# B&R Automation Studio project SDCAxis
Automation Studio 4.5.2.102; Default project; technology packages: Acp10Arnc0 1.0.0

## Configuration Real

CPU 4PP065.0571-P74, AutomationRuntime D4.52, Build 4.1.2, Vc V4.25.0, Safety 1.6

### Task classes (Cpu.sw)
```
Cyclic#1 (cycle 2000 us, tolerance 0 us):
  SDCAxisCtr <- SDCAxisCtrl_X.prg
DataObjects: Arnc0sys
NcDataObjects: AxisInit <- AxisInit.dob, gAxis03a <- gAxis03obj.gAxis03a.dob, AxisApt <- AxisApt.dob, gAxis03i <- gAxis03obj.gAxis03i.dob
Binaries: TCData, Acp10map1, acp10cfg, Acp10map, arconfig, User, Role, sysconf, iomap, asfw, ashwd, arnc0cfg, Arnc0map
Libraries: Acp10sdc, Library, Acp10man, Acp10_MC, sys_lib, brsystem, asstring, powerlnk, asieccon, AsMath, Arnc0man, DataObj, AsArLog, FileIO, AsArProf, AsMem, Runtime, astime, Acp10par, NcGlobal, asiotime
```

### Hardware
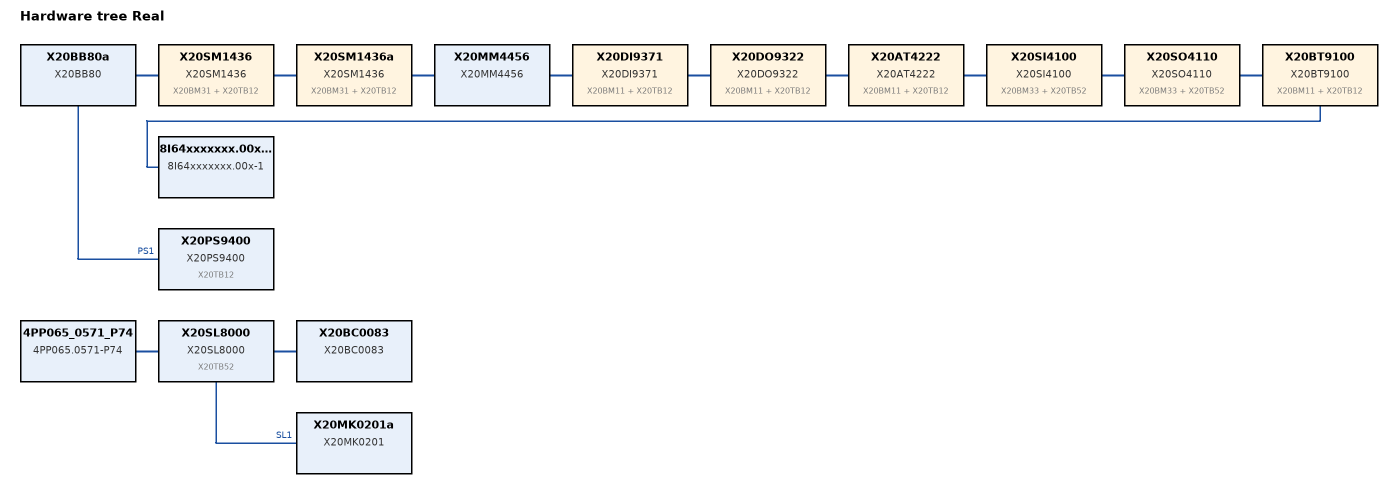
```
4PP065_0571_P74 : 4PP065.0571-P74 v1.1.2.0
  Connector IF4:
    EplInterfaceRedundant = 0
    EplEthInterfaceRedundant = 0
  Connector IF5:
    ActivateDevice = 1
    Mode = Manual
    InternetAddress = 10.0.1.14
    SubnetMask = 255.255.255.0
  ConfigurationID = labBR
  TimerDeviceType = EPLX2X
  TimerDevice = 4PP065_0571_P74.IF4
  TaskClassIdleTime = 2000
  Cyclic1Duration = 2000
  Cyclic1Tolerance = 0
  Cyclic1Output = 1
  Cyclic3Tolerance = 0
  VcObjectName = Visu
8I64xxxxxxx.00x-1 : 8I64xxxxxxx.00x-1 v1.3.9.1  [X2X1 -> X20BT9100.X2X1 [Cable Type=X2XCable, Length=10, Version=1.0.0.2]]
  BothEndSwitchesAreNormallyOpen_r1 = on
  QuickStopIsNormallyOpen_r1 = on
X20AT4222 : X20AT4222 v1.2.3.0  [SS1 -> X20TB12f.SS; SL -> X20BM11c.SL1]
X20BB80a : X20BB80 v1.0.2.0
X20BC0083 : X20BC0083 v2.7.0.0  [PLK1 -> X20SL8000.PLK2 (NodeNumber=2) [Cable Type=PowerlinkCable, Length=10, Version=1.0.0.2]; SL -> X20BB80a.SL1]
X20BM11a : X20BM11 v1.0.0.1  [X2X1 -> X20MM4456.X2X2]
X20BM11b : X20BM11 v1.0.0.1  [X2X1 -> X20BM11a.X2X2]
X20BM11c : X20BM11 v1.0.0.1  [X2X1 -> X20BM11b.X2X2]
X20BM11d : X20BM11 v1.0.0.1  [X2X1 -> X20BM33b.X2X2]
X20BM31a : X20BM31 v1.0.0.1  [X2X1 -> X20BB80a.IF1]
X20BM31b : X20BM31 v1.0.0.1  [X2X1 -> X20BM31a.X2X2]
X20BM33a : X20BM33 v1.0.0.4  [X2X1 -> X20BM11c.X2X2]
X20BM33b : X20BM33 v1.0.0.4  [X2X1 -> X20BM33a.X2X2]
X20BT9100 : X20BT9100 v1.0.3.0  [SS1 -> X20TB12g.SS; SL -> X20BM11d.SL1]
X20DI9371 : X20DI9371 v1.0.2.0  [SS1 -> X20TB12d.SS; SL -> X20BM11a.SL1]
X20DO9322 : X20DO9322 v1.0.3.0  [SS1 -> X20TB12e.SS; SL -> X20BM11b.SL1]
X20MK0201a : X20MK0201 v1.0.0.0  [SL -> X20SL8000.SL1]
X20MM4456 : X20MM4456 v1.1.5.0  [X2X1 -> X20BM31b.X2X2]
X20PS9400 : X20PS9400 v1.0.2.4  [SS1 -> X20TB12b.SS; PS -> X20BB80a.PS1]
X20SI4100 : X20SI4100 v1.10.1.1  [SS1 -> X20TB52b.SS; SL -> X20BM33a.SL1]
X20SL8000 : X20SL8000 v1.6.5.1  [PLK1 -> 4PP065_0571_P74.IF4 (NodeNumber=1) [Cable Type=PowerlinkCable, Length=10, Version=1.0.0.2]; PLK2 -> X20BC0083.PLK1 (NodeNumber=1) [Cable Type=PowerlinkCable, Length=10, Version=1.0.0.2]; SS1 -> X20TB52a.SS]
  SafeProject = SafeLOGIC-1
X20SM1436 : X20SM1436 v1.4.2.1  [SS1 -> X20TB12a.SS; SL -> X20BM31a.SL1]
X20SM1436a : X20SM1436 v1.4.2.1  [SS1 -> X20TB12c.SS; SL -> X20BM31b.SL1]
X20SO4110 : X20SO4110 v1.10.1.1  [SS1 -> X20TB52c.SS; SL -> X20BM33b.SL1]
  SafeLogicID = 2
  SafeModuleID = 3
X20TB12a : X20TB12 v1.0.0.0
X20TB12b : X20TB12 v1.0.0.0
X20TB12c : X20TB12 v1.0.0.0
X20TB12d : X20TB12 v1.0.0.0
X20TB12e : X20TB12 v1.0.0.0
X20TB12f : X20TB12 v1.0.0.0
X20TB12g : X20TB12 v1.0.0.0
X20TB52a : X20TB52 v1.0.0.1
X20TB52b : X20TB52 v1.0.0.1
X20TB52c : X20TB52 v1.0.0.1
```

### IoMap.iom - 4PP065_0571_P74/IoMap.iom
```iecst
VAR_CONFIG
	Cyclic#1.gAxis03_DrvIf.iLifeCnt AT %IB."8I64xxxxxxx.00x-1".SDC_LifeCnt;
	Cyclic#1.gAxis03_DrvIf.iDrvOK AT %IX."8I64xxxxxxx.00x-1".ETAD_Input_Bool_02;
	Cyclic#1.gAxis03_DrvIf.oSetTime AT %QW."8I64xxxxxxx.00x-1".SDC_SetTime;
	Cyclic#1.gAxis03_DrvIf.oSetPos AT %QW."8I64xxxxxxx.00x-1".LFRD_Output;
	Cyclic#1.gAxis03_DiDoIf.iLifeCntDriveReady AT %IB."8I64xxxxxxx.00x-1".SDC_LifeCnt;
	Cyclic#1.gAxis03_DiDoIf.iLifeCntDriveEnable AT %IB."8I64xxxxxxx.00x-1".SDC_LifeCnt;
	Cyclic#1.gAxis03_DiDoIf.oDriveEnable AT %QX."8I64xxxxxxx.00x-1".CMDD_Output_Bool_00;
	Cyclic#1.gAxis03_ModuleOk AT %QX."8I64xxxxxxx.00x-1".CMDD_Output_Bool_01;
	Cyclic#1.gAxis03_ModuleOk AT %QX."8I64xxxxxxx.00x-1".CMDD_Output_Bool_02;
	Cyclic#1.gAxis03_ModuleOk AT %IX."8I64xxxxxxx.00x-1".ModuleOk;
	Cyclic#1.gAxis03_DiDoIf.oDriveEnable AT %QX."8I64xxxxxxx.00x-1".CMDD_Output_Bool_03;
	Cyclic#1.gAxis03_DiDoIf.iDriveReady AT %IX."8I64xxxxxxx.00x-1".ETAD_Input_Bool_02;
	::SDCAxisCtr:pwm_period AT %QW."X20MM4456".PeriodDurationPWM;
	::SDCAxisCtr:coil_pwm_value AT %QW."X20MM4456".PulseWidthCurrentPWM04;
	::SDCAxisCtr:axis_X.pwm_value AT %QW."X20MM4456".PulseWidthCurrentPWM01;
	::SDCAxisCtr:axis_X.reset_error AT %QX."X20MM4456".ClearError01;
	::SDCAxisCtr:axis_X.reset_counter AT %QX."X20MM4456".ResetCounter01;
	::SDCAxisCtr:axis_X.counter AT %IW."X20MM4456".Counter01;
	::SDCAxisCtr:coil_powered AT %IX."X20DI9371".DigitalInput01;
	::SDCAxisCtr:axis_X.endswitch_a_reached AT %IX."X20MM4456".StatusInput03;
	::SDCAxisCtr:axis_X.endswitch_b_reached AT %IX."X20MM4456".StatusInput04;
END_VAR
```

### Acp10cfg.ncc - 4PP065_0571_P74/Motion/Acp10cfg.ncc
```
NcConfiguration (Version=3.13.1, NcSwId=Acp10)
  ACP10CF1_typ:
    cnt_nettrc_rec_drive = 1500
    bufsize_trace_upload = 1200
    tc_nc_man_task = Cyclic #1
    glob_pv_as_ncobject = Yes
    ncsys_dl_broadcast = Yes
    ncsys_dl_acp_reset = Yes
    safemc_log_err_to_ax = Yes
    network_init:
      ncsw_init_execute = Yes
      automatic_execute = No
      node_nr_warning = Yes
      net_err_before_ncact = Yes
    nettrc:
      enter_parsecrec = Yes
      enter_ncaction = Yes
      save_ring_startidx = Yes
    cam_prof_download:
      cam_dat_dl_parallel = No
      tc_cam_dl_parallel = Task class for NC Manager task
    sdc_if[0]:
      if_name = SDC_IF1
      mc_broadcast_size = 800
      mc_broadcast_extdat = No
```

### Acp10map.ncm - 4PP065_0571_P74/Motion/Acp10map.ncm
```
NcMapping (NcSwId=Acp10, DisabledNodesAreHidden=False)
  NcObject gAxis03 (ModuleId=8I64xxxxxxx.00x-1, ModuleAddress=SDC_IF1.ST1, Type=ncAXIS, Channel=1, AcoposSimulation=Off, InitParameter=gAxis03i, AcoposParameter=gAxis03a, AdditionalData=CNC_Enabled="1" , Disabled=FALSE, ModuleDisabled=FALSE)
```

### Acp10map1.ncm - 4PP065_0571_P74/Motion/Acp10map1.ncm
```
NcMapping (NcSwId=ACP10, DisabledNodesAreHidden=False)
  NcObject AxisX (ModuleAddress=SDC_IF1.ST2, InterfaceType=SDC, Type=ncAXIS, Channel=1, AcoposSimulation=Off, InitParameter=gAxis03i, AcoposParameter=gAxis03a, AdditionalData=CNC_Enabled="1" , Disabled=FALSE, ModuleDisabled=FALSE)
  NcObject AxisY (ModuleAddress=SDC_IF1.ST3, InterfaceType=SDC, Type=ncAXIS, Channel=1, AcoposSimulation=Off, InitParameter=AxisInit, AcoposParameter=AxisApt, AdditionalData=CNC_Enabled="1" , Disabled=FALSE)
  NcObject AxisZ (ModuleAddress=SDC_IF1.ST4, InterfaceType=SDC, Type=ncAXIS, Channel=1, AcoposSimulation=Off, InitParameter=AxisInit, AcoposParameter=AxisApt, AdditionalData=CNC_Enabled="1" , Disabled=FALSE)
```

### Arnc0cfg.ncc - 4PP065_0571_P74/Motion/Arnc0cfg.ncc
```
NcConfiguration (Version=3.13.1, NcSwId=Arnc0)
  ARNC0CFG_typ:
    sampling_rate = 4000
    cnt_nettrc_rec_drive = 150
    bufsize_sys_trace = 16#00005000
    enable_mp_log = Yes
    tc_nc_man_task = Cyclic #1
    bg_load = 1
    glob_pv_as_ncobject = Yes
```

### Arnc0map.ncm - 4PP065_0571_P74/Motion/Arnc0map.ncm
```
NcMapping (NcSwId=Arnc0, DisabledNodesAreHidden=False)
  NcObject CNCsys (Type=ncCNCSYS, Channel=1, AcoposSimulation=Off, InitParameter=CncInit, Disabled=FALSE, ModuleDisabled=FALSE)
  NcObject CNC2 (Type=ncCNCSYS, Channel=2, AcoposSimulation=Off, Disabled=TRUE, ModuleDisabled=FALSE)
  NcObject CNC3 (Type=ncCNCSYS, Channel=3, AcoposSimulation=Off, Disabled=TRUE, ModuleDisabled=FALSE)
  NcObject CNC4 (Type=ncCNCSYS, Channel=4, AcoposSimulation=Off, Disabled=TRUE, ModuleDisabled=FALSE)
  NcObject CNC5 (Type=ncCNCSYS, Channel=5, AcoposSimulation=Off, Disabled=TRUE, ModuleDisabled=FALSE)
  NcObject CNC6 (Type=ncCNCSYS, Channel=6, AcoposSimulation=Off, Disabled=TRUE, ModuleDisabled=FALSE)
  NcObject CNC7 (Type=ncCNCSYS, Channel=7, AcoposSimulation=Off, Disabled=TRUE, ModuleDisabled=FALSE)
  NcObject CNC8 (Type=ncCNCSYS, Channel=8, AcoposSimulation=Off, Disabled=TRUE, ModuleDisabled=FALSE)
  NcObject CNC9 (Type=ncCNCSYS, Channel=9, AcoposSimulation=Off, Disabled=TRUE, ModuleDisabled=FALSE)
  NcObject CNC10 (Type=ncCNCSYS, Channel=10, AcoposSimulation=Off, Disabled=TRUE, ModuleDisabled=FALSE)
  NcObject CNC11 (Type=ncCNCSYS, Channel=11, AcoposSimulation=Off, Disabled=TRUE, ModuleDisabled=FALSE)
  NcObject CNC12 (Type=ncCNCSYS, Channel=12, AcoposSimulation=Off, Disabled=TRUE, ModuleDisabled=FALSE)
  NcObject CNC13 (Type=ncCNCSYS, Channel=13, AcoposSimulation=Off, Disabled=TRUE, ModuleDisabled=FALSE)
  NcObject CNC14 (Type=ncCNCSYS, Channel=14, AcoposSimulation=Off, Disabled=TRUE, ModuleDisabled=FALSE)
  NcObject CNC15 (Type=ncCNCSYS, Channel=15, AcoposSimulation=Off, Disabled=TRUE, ModuleDisabled=FALSE)
  NcObject CNC16 (Type=ncCNCSYS, Channel=16, AcoposSimulation=Off, Disabled=TRUE, ModuleDisabled=FALSE)
  NcObject CNC17 (Type=ncCNCSYS, Channel=17, AcoposSimulation=Off, Disabled=TRUE, ModuleDisabled=FALSE)
  NcObject CNC18 (Type=ncCNCSYS, Channel=18, AcoposSimulation=Off, Disabled=TRUE, ModuleDisabled=FALSE)
  NcObject CNC19 (Type=ncCNCSYS, Channel=19, AcoposSimulation=Off, Disabled=TRUE, ModuleDisabled=FALSE)
  NcObject CNC20 (Type=ncCNCSYS, Channel=20, AcoposSimulation=Off, Disabled=TRUE, ModuleDisabled=FALSE)
  NcObject CNC21 (Type=ncCNCSYS, Channel=21, AcoposSimulation=Off, Disabled=TRUE, ModuleDisabled=FALSE)
  NcObject CNC22 (Type=ncCNCSYS, Channel=22, AcoposSimulation=Off, Disabled=TRUE, ModuleDisabled=FALSE)
  NcObject CNC23 (Type=ncCNCSYS, Channel=23, AcoposSimulation=Off, Disabled=TRUE, ModuleDisabled=FALSE)
  NcObject CNC24 (Type=ncCNCSYS, Channel=24, AcoposSimulation=Off, Disabled=TRUE, ModuleDisabled=FALSE)
```

## Configuration Simulation

CPU , AutomationRuntime J4.25, Safety 1.10

### Task classes (Cpu.sw)
```
Cyclic#1 (cycle 2000 us, tolerance 0 us):
  SDCAxisCtr <- SDCAxisCtrl_X.prg
  ncsdcctrl <- ncsdcctrl.prg
DataObjects: Acp10sys
NcDataObjects: AxisApt <- AxisApt.dob, AxisInit <- AxisInit.dob, acp10etxen <- acp10etxen.dob, gAxis05a <- gAxis05obj.gAxis05a.dob, gAxis05i <- gAxis05obj.gAxis05i.dob
Binaries: TCData, ashwd, sysconf, asfw, arconfig, iomap, Acp10map, Acp10map1, arnc0cfg, acp10cfg
Libraries: AsIecCon, astime, Acp10sdc, Acp10man, Acp10par, NcGlobal, asstring, AsIOTime, Acp10_MC, brsystem, sys_lib, Runtime, Acp10sim, fileio, powerlnk, Library, AsBrStr
```

### Hardware
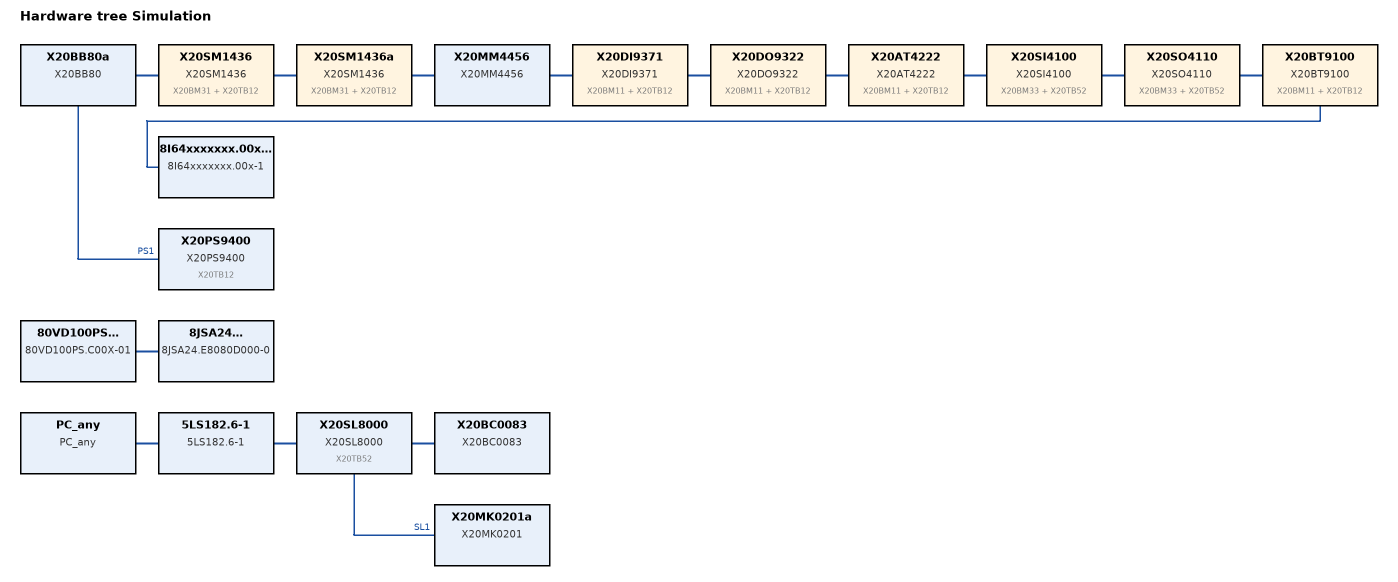
```
5LS182.6-1 : 5LS182.6-1 v1.3.0.0  [SL -> PC_any.SL1]
80VD100PS.C00X-01 : 80VD100PS.C00X-01 v2.3.0.1
8I64xxxxxxx.00x-1 : 8I64xxxxxxx.00x-1 v1.3.9.1  [X2X1 -> X20BT9100.X2X1 [Cable Type=X2XCable, Length=10, Version=1.0.0.2]]
  BothEndSwitchesAreNormallyOpen_r1 = on
  QuickStopIsNormallyOpen_r1 = on
8JSA24.E8080D000-0 : 8JSA24.E8080D000-0 v1.0.6.30  [MT -> 80VD100PS.C00X-01.MT1]
PC_any : PC_any v1.1.0.0 (OrderNumber=PC)
  ConfigurationID = SDCAxis_Simulation
  SystemTick = 2000
  Cyclic1Duration = 2000
  Cyclic1Tolerance = 0
  Cyclic1Output = 1
X20AT4222 : X20AT4222 v1.2.3.0  [SS1 -> X20TB12f.SS; SL -> X20BM11c.SL1]
X20BB80a : X20BB80 v1.0.2.0
X20BC0083 : X20BC0083 v2.7.0.0  [PLK2 -> X20SL8000.PLK2 (NodeNumber=2) [Cable Type=PowerlinkCable, Length=10, Version=1.0.0.2]; SL -> X20BB80a.SL1]
X20BM11a : X20BM11 v1.0.0.1  [X2X1 -> X20MM4456.X2X2]
X20BM11b : X20BM11 v1.0.0.1  [X2X1 -> X20BM11a.X2X2]
X20BM11c : X20BM11 v1.0.0.1  [X2X1 -> X20BM11b.X2X2]
X20BM11d : X20BM11 v1.0.0.1  [X2X1 -> X20BM33b.X2X2]
X20BM31a : X20BM31 v1.0.0.1  [X2X1 -> X20BB80a.IF1]
X20BM31b : X20BM31 v1.0.0.1  [X2X1 -> X20BM31a.X2X2]
X20BM33a : X20BM33 v1.0.0.4  [X2X1 -> X20BM11c.X2X2]
X20BM33b : X20BM33 v1.0.0.4  [X2X1 -> X20BM33a.X2X2]
X20BT9100 : X20BT9100 v1.0.3.0  [SS1 -> X20TB12g.SS; SL -> X20BM11d.SL1]
X20DI9371 : X20DI9371 v1.0.2.0  [SS1 -> X20TB12d.SS; SL -> X20BM11a.SL1]
X20DO9322 : X20DO9322 v1.0.3.0  [SS1 -> X20TB12e.SS; SL -> X20BM11b.SL1]
X20MK0201a : X20MK0201 v1.0.0.0  [SL -> X20SL8000.SL1]
X20MM4456 : X20MM4456 v1.1.5.0  [X2X1 -> X20BM31b.X2X2]
X20PS9400 : X20PS9400 v1.0.2.4  [SS1 -> X20TB12b.SS; PS -> X20BB80a.PS1]
X20SI4100 : X20SI4100 v1.10.1.1  [SS1 -> X20TB52b.SS; SL -> X20BM33a.SL1]
X20SL8000 : X20SL8000 v1.6.5.1  [PLK1 -> 5LS182.6-1.IF1 (NodeNumber=1) [Cable Type=PowerlinkCable, Length=10, Version=1.0.0.2]; PLK2 -> X20BC0083.PLK2 (NodeNumber=1) [Cable Type=PowerlinkCable, Length=10, Version=1.0.0.2]; SS1 -> X20TB52a.SS]
  SafeProject = SafeLOGIC-1
X20SM1436 : X20SM1436 v1.4.2.1  [SS1 -> X20TB12a.SS; SL -> X20BM31a.SL1]
X20SM1436a : X20SM1436 v1.4.2.1  [SS1 -> X20TB12c.SS; SL -> X20BM31b.SL1]
X20SO4110 : X20SO4110 v1.10.1.1  [SS1 -> X20TB52c.SS; SL -> X20BM33b.SL1]
  SafeLogicID = 2
  SafeModuleID = 3
X20TB12a : X20TB12 v1.0.0.0
X20TB12b : X20TB12 v1.0.0.0
X20TB12c : X20TB12 v1.0.0.0
X20TB12d : X20TB12 v1.0.0.0
X20TB12e : X20TB12 v1.0.0.0
X20TB12f : X20TB12 v1.0.0.0
X20TB12g : X20TB12 v1.0.0.0
X20TB52a : X20TB52 v1.0.0.1
X20TB52b : X20TB52 v1.0.0.1
X20TB52c : X20TB52 v1.0.0.1
```

### IOMap.iom - PC_any/IOMap.iom
```iecst
VAR_CONFIG
	::SDCAxisCtr:pwm_period AT %QW."X20MM4456".PeriodDurationPWM;
	::SDCAxisCtr:coil_pwm_value AT %QW."X20MM4456".PulseWidthCurrentPWM04;
	::SDCAxisCtr:axis_X.pwm_value AT %QW."X20MM4456".PulseWidthCurrentPWM01;
	::SDCAxisCtr:axis_X.reset_error AT %QX."X20MM4456".ClearError01;
	::SDCAxisCtr:axis_X.reset_counter AT %QX."X20MM4456".ResetCounter01;
	::SDCAxisCtr:axis_X.counter AT %IW."X20MM4456".Counter01;
	::SDCAxisCtr:axis_X.endswitch_a_reached AT %IX."X20MM4456".StatusInput03; (*Logical condition input 01=Motor 01:A*)
	::SDCAxisCtr:axis_X.endswitch_b_reached AT %IX."X20MM4456".StatusInput04; (*Logical condition input 02=Motor 01:B*)
	::SDCAxisCtr:coil_powered AT %IX."X20DI9371".DigitalInput01;
	Cyclic#1.gAxis03_DrvIf.iLifeCnt AT %IB."8I64xxxxxxx.00x-1".SDC_LifeCnt;
	Cyclic#1.gAxis03_DrvIf.iDrvOK AT %IX."8I64xxxxxxx.00x-1".ETAD_Input_Bool_02;
	Cyclic#1.gAxis03_DrvIf.oSetTime AT %QW."8I64xxxxxxx.00x-1".SDC_SetTime;
	Cyclic#1.gAxis03_DrvIf.oSetPos AT %QW."8I64xxxxxxx.00x-1".LFRD_Output;
	Cyclic#1.gAxis03_DiDoIf.iLifeCntDriveReady AT %IB."8I64xxxxxxx.00x-1".SDC_LifeCnt;
	Cyclic#1.gAxis03_DiDoIf.iLifeCntDriveEnable AT %IB."8I64xxxxxxx.00x-1".SDC_LifeCnt;
	Cyclic#1.gAxis03_DiDoIf.oDriveEnable AT %QX."8I64xxxxxxx.00x-1".CMDD_Output_Bool_00;
	Cyclic#1.gAxis03_ModuleOk AT %QX."8I64xxxxxxx.00x-1".CMDD_Output_Bool_01;
	Cyclic#1.gAxis03_ModuleOk AT %QX."8I64xxxxxxx.00x-1".CMDD_Output_Bool_02;
	Cyclic#1.gAxis03_ModuleOk AT %IX."8I64xxxxxxx.00x-1".ModuleOk;
	Cyclic#1.gAxis03_DiDoIf.oDriveEnable AT %QX."8I64xxxxxxx.00x-1".CMDD_Output_Bool_03;
	Cyclic#1.gAxis03_DiDoIf.iDriveReady AT %IX."8I64xxxxxxx.00x-1".ETAD_Input_Bool_02;
	      Cyclic#1.gAxis05_DrvIf.iLifeCnt AT %IB."X20SM1436".LifeCnt;
	      Cyclic#1.gAxis05_DrvIf.iDrvOK AT %IX."X20SM1436".DrvOk01;
	      Cyclic#1.gAxis05_DrvIf.oBoostCurrent AT %QX."X20SM1436".BoostCurrent01;
	      Cyclic#1.gAxis05_DrvIf.oStandStillCurrent AT %QX."X20SM1436".StandstillCurrent01;
	      Cyclic#1.gAxis05_DrvIf.oSetTime AT %QW."X20SM1436".SetTime01;
	      Cyclic#1.gAxis05_MotorStep0 AT %QW."X20SM1436".Motor1Step0;
	      Cyclic#1.gAxis05_DiDoIf.iLifeCntDriveEnable AT %IB."X20SM1436".LifeCnt;
	      Cyclic#1.gAxis05_DiDoIf.iLifeCntDriveReady AT %IB."X20SM1436".LifeCnt;
	      Cyclic#1.gAxis05_DiDoIf.iDriveReady AT %IX."X20SM1436".DrvOk01;
	      Cyclic#1.gAxis05_DiDoIf.oDriveEnable AT %QX."X20SM1436".DriveEnable01;
	      Cyclic#1.gAxis05_EncIf1.iLifeCnt AT %IB."X20SM1436".LifeCnt;
	      Cyclic#1.gAxis05_EncIf1.iEncOK AT %IX."X20SM1436".EncOk01;
	      Cyclic#1.gAxis05_EncIf1.iActPos AT %IW."X20SM1436".ActPos01;
	      Cyclic#1.gAxis05_EncIf1.iRefPulsePos AT %IW."X20SM1436".RefPulsePos01;
	      Cyclic#1.gAxis05_EncIf1.iRefPulseCnt AT %IB."X20SM1436".RefPulseCnt01;
	      Cyclic#1.gAxis05_EncIf1.iActTime AT %IW."X20SM1436".ActTime01;
END_VAR
```

### Acp10cfg.ncc - PC_any/Motion/Acp10cfg.ncc
```
NcConfiguration (Version=3.13.1, NcSwId=Acp10)
  ACP10CF1_typ:
    cnt_nettrc_rec_drive = 150
    bufsize_trace_upload = 1200
    tc_nc_man_task = Cyclic #1
    glob_pv_as_ncobject = Yes
    ncsys_dl_broadcast = Yes
    ncsys_dl_acp_reset = Yes
    safemc_log_err_to_ax = Yes
    network_init:
      ncsw_init_execute = Yes
      automatic_execute = No
      node_nr_warning = Yes
      net_err_before_ncact = Yes
    nettrc:
      enter_parsecrec = Yes
      enter_ncaction = Yes
      save_ring_startidx = No
    cam_prof_download:
      cam_dat_dl_parallel = No
      tc_cam_dl_parallel = Task class for NC Manager task
    sdc_if[0]:
      if_name = SDC_IF1
      mc_broadcast_size = 800
      mc_broadcast_extdat = No
```

### Acp10map.ncm - PC_any/Motion/Acp10map.ncm
```
NcMapping (NcSwId=Acp10)
  NcObject gAxis04 (ModuleId=8I64xxxxxxx.00x-1, ModuleAddress=SDC_IF1.ST2, Type=ncAXIS, Channel=1, AcoposSimulation=Off, InitParameter=gAxis03i, AcoposParameter=gAxis03a, AdditionalData=CNC_Enabled="1" , Disabled=FALSE, ModuleDisabled=FALSE)
  NcObject gAxis05 (ModuleId=X20SM1436, ModuleAddress=SDC_IF1.ST3, Type=ncAXIS, Channel=1, AcoposSimulation=Off, InitParameter=gAxis05i, AcoposParameter=gAxis05a, Disabled=FALSE, ModuleDisabled=FALSE)
  NcObject X20SM1436a_ncAXIS1 (ModuleId=X20SM1436a, ModuleAddress=SDC_IF1.ST4, Type=ncAXIS, Channel=1, AcoposSimulation=Off, Disabled=TRUE, ModuleDisabled=FALSE)
```

### Acp10map1.ncm - PC_any/Motion/Acp10map1.ncm
```
NcMapping (NcSwId=ACP10, DisabledNodesAreHidden=False)
  NcObject MyLittleAxis (ModuleAddress=SDC_IF1.ST1, InterfaceType=SDC, Type=ncAXIS, Channel=1, AcoposSimulation=Off, InitParameter=MyLittleIn, AcoposParameter=MyLittleAp, Disabled=FALSE, ModuleDisabled=FALSE)
```

### Arnc0cfg.ncc - PC_any/Motion/Arnc0cfg.ncc
```
NcConfiguration (Version=1.45.0, NcSwId=ARNC0)
  ARNC0CFG_typ:
    sampling_rate = 4000
    cnt_nettrc_rec_drive = 150
    bufsize_sys_trace = 16#00005000
    enable_mp_log = Yes
    tc_nc_man_task = Cyclic #1
    bg_load = 1
    glob_pv_as_ncobject = Yes
```

## Logical view

Binary libraries used (declarations not repeated): Runtime, OPERATOR, AsIecCon, astime, Acp10sdc 3.13.1, Acp10man 3.13.1, Acp10par 3.13.1, NcGlobal 3.13.1, asstring, AsIOTime, Acp10_MC 3.13.1, brsystem, sys_lib, Acp10sim 3.13.1, AsMath, Arnc0man 3.13.0, DataObj, AsArLog, FileIO, AsArProf, AsMem, AsBrStr

### Global.var - Global variables
```iecst
VAR
	AxisX : ACP10AXIS_typ := (0);
	AxisX_EncIf : SdcEncIf16_typ := (0);
	AxisX_DrvIf : SdcDrvIf16_typ := (0);
	AxisX_DiDoIf : SdcDiDoIf_typ := (0);
	AxisX_HW : SdcHwCfg_typ := (0);
	gAxis01 : ACP10AXIS_typ := (0);
	gAxis02 : ACP10AXIS_typ := (0);
	gAxisTest : ACP10AXIS_typ := (0);
	gAxisTest_HW : SdcHwCfg_typ := (0);
	gAxisTest_DrvIf : SdcDrvIf16_typ := (0);
	gAxisTest_DiDoIf : SdcDiDoIf_typ := (0);
	gAxisTest_ModuleOk : BOOL := 0;
	gAxis03 : ACP10AXIS_typ := (0);
	gAxis03_HW : SdcHwCfg_typ := (0);
	gAxis03_DrvIf : SdcDrvIf16_typ := (0);
	gAxis03_DiDoIf : SdcDiDoIf_typ := (0);
	gAxis03_ModuleOk : BOOL := 0;
	CNCsys : ARNC0CNC_typ;
	gAxis04 : ACP10AXIS_typ := (0);
	gAxis05 : ACP10AXIS_typ := (0);
	gAxis05_HW : SdcHwCfg_typ := (0);
	gAxis05_DrvIf : SdcDrvIf16_typ := (0);
	gAxis05_EncIf1 : SdcEncIf16_typ := (0);
	gAxis05_DiDoIf : SdcDiDoIf_typ := (0);
	gAxis05_MotorStep0 : INT := 0;
	coil_powered : BOOL := FALSE;
	coil_pwm_value : INT := 0;
	fb_regulator : FB_Regulator;
	pwm_period : UINT := 0;
	axis_X : FB_Axis := (0);
	iPosHwEnd : BOOL := FALSE;
	iNegHwEnd : BOOL := FALSE;
	iActPos : USINT := 0;
	oSetPos : USINT := 0;
END_VAR
```

### Package Logical/Libraries - Global libraries

### Library Logical/Libraries/Library (ANSIC)

#### Library.fun
```iecst
FUNCTION_BLOCK FB_Motor (*TODO: Add your comment here*) (*$GROUP=User,$CAT=User,$GROUPICON=User.png,$CATICON=User.png*)
	VAR_INPUT
		in : REAL;
	END_VAR
	VAR_OUTPUT
		out_w : REAL;
		out_phi : REAL;
	END_VAR
	VAR
		k_e : REAL;
		T_m : REAL;
		dt : REAL;
		integrator : FB_Integrator;
		integrator_phi : FB_Integrator;
	END_VAR
END_FUNCTION_BLOCK

FUNCTION_BLOCK FB_Integrator (*TODO: Add your comment here*) (*$GROUP=User,$CAT=User,$GROUPICON=User.png,$CATICON=User.png*)
	VAR_INPUT
		in : REAL;
		dt : REAL;
	END_VAR
	VAR_OUTPUT
		out : REAL;
	END_VAR
	VAR
		state : REAL := 0.0;
	END_VAR
END_FUNCTION_BLOCK

FUNCTION_BLOCK FB_Controller (* *) (*$GROUP=User,$CAT=User,$GROUPICON=User.png,$CATICON=User.png*)
	VAR_INPUT
		in : REAL;
	END_VAR
	VAR_OUTPUT
		out : REAL;
	END_VAR
	VAR
		k_i : REAL;
		sum : REAL;
		k_p : REAL;
		dt : REAL;
		max_abs_value : REAL;
		integrator : FB_Integrator;
		last_sum : REAL;
	END_VAR
END_FUNCTION_BLOCK

FUNCTION_BLOCK FB_Endswitch (*TODO: Add your comment here*) (*$GROUP=User,$CAT=User,$GROUPICON=User.png,$CATICON=User.png*)
	VAR_INPUT
		in : REAL;
		neg_value : REAL;
		pos_value : REAL;
	END_VAR
	VAR_OUTPUT
		neg_reached : BOOL;
		pos_reached : BOOL;
	END_VAR
END_FUNCTION_BLOCK

FUNCTION_BLOCK FB_Axis (*TODO: Add your comment here*) (*$GROUP=User,$CAT=User,$GROUPICON=User.png,$CATICON=User.png*)
	VAR_INPUT
		u : REAL;
		reset_error : BOOL;
		endswitch_a_reached : BOOL;
		endswitch_b_reached : BOOL;
		pwm_percentage : SINT;
	END_VAR
	VAR_OUTPUT
		reset_counter : BOOL;
		pwm_value : INT;
	END_VAR
	VAR_OUTPUT RETAIN
		counter : INT;
	END_VAR
	VAR_OUTPUT
		speed : REAL;
	END_VAR
	VAR
		i : INT;
		last_counter : INT;
		dir : BOOL;
		spid : REAL;
		k : INT;
	END_VAR
END_FUNCTION_BLOCK

{REDUND_ERROR} FUNCTION_BLOCK FB_Regulator (*TODO: Add your comment here*) (*$GROUP=User,$CAT=User,$GROUPICON=User.png,$CATICON=User.png*)
	VAR_INPUT
		e : REAL;
	END_VAR
	VAR_OUTPUT
		u : REAL;
	END_VAR
	VAR
		k_p : REAL;
		k_i : REAL;
		integrator : FB_Integrator;
		iyOld : REAL;
		max_abc_value : REAL := 24;
		dt : REAL;
		x : REAL;
	END_VAR
END_FUNCTION_BLOCK
```

#### FB_Motor.c
```c
#include <bur/plctypes.h>
#ifdef __cplusplus
	extern "C"
	{
#endif
	#include "Library.h"
#ifdef __cplusplus
	};
#endif
/* TODO: Add your comment here */
void FB_Motor(struct FB_Motor* inst)
{/*
	inst->integrator.in = (inst->u/inst->ke - inst->w) * (inst->dt/inst->Tm);
	FB_Integrator(&inst->integrator);
	inst->w = inst->integrator.out;
	inst->integrator.in = inst->w * inst->dt;
	FB_Integrator(&inst->integrator);
	inst->phi = inst->integrator.out;*/
}
```

#### FB_Controller.c
```c
#include <bur/plctypes.h>
#ifdef __cplusplus
	extern "C"
	{
#endif
	#include "Library.h"
#ifdef __cplusplus
	};
#endif

void FB_Controller(struct FB_Controller* inst)
{

}
```

#### FB_Integrator.c
```c
#include <bur/plctypes.h>
#ifdef __cplusplus
	extern "C"
	{
#endif
	#include "Library.h"
#ifdef __cplusplus
	};
#endif
/* TODO: Add your comment here */
void FB_Integrator(struct FB_Integrator* inst)
{
	inst->out = inst->dt * inst->in + inst->state;
	inst->state = inst->out;
}
```

#### FB_Endswitch.c
```c
#include <bur/plctypes.h>
#ifdef __cplusplus
	extern "C"
	{
#endif
	#include "Library.h"
#ifdef __cplusplus
	};
#endif
/* TODO: Add your comment here */
void FB_Endswitch(struct FB_Endswitch* inst)
{

}
```

#### FB_Axis.c
```c
#include <bur/plctypes.h>
#ifdef __cplusplus
	extern "C"
	{
#endif
	#include "Library.h"
#ifdef __cplusplus
	};
#endif
/* TODO: Add your comment here */
void FB_Axis(struct FB_Axis* inst)
{
	if (inst->endswitch_a_reached == 1 )
	{
		inst->dir = 1;
	}
	if (inst->endswitch_b_reached == 1 )
	{
		inst->dir = 0;
	}

	if(inst->dir == 1)
	{
		//inst->reset_counter = 0;
		inst->u = -inst->u;
		inst->pwm_value = (inst->u/24.0) * 32767;
	}
	if(inst->dir == 0)
	{
		//inst->reset_counter = 0;
		inst->pwm_value = (inst->u/24.0) * 32767;
	}
	if (inst->i == 1000)
	{
		inst->speed = (inst->counter - inst->last_counter)/2;
		inst->last_counter = inst->counter;
		inst->i = 0;
	}
	inst->spid = inst->speed;
	inst->i++;
}
```

#### FB_Regulator.c
```c
#include <bur/plctypes.h>
#ifdef __cplusplus
	extern "C"
	{
#endif
	#include "Library.h"
#ifdef __cplusplus
	};
#endif
/* TODO: Add your comment here */
void FB_Regulator(struct FB_Regulator* inst)
{
	float BON(float x)
		{
		if(x < 0)
		{
			if(x < -inst->max_abc_value)
				return -inst->max_abc_value;
			else
				return x;
		}
		else
		{
			if(x > inst->max_abc_value)
				return inst->max_abc_value;
			else
				return x;
		}

	}
	inst->integrator.in = inst->e * inst->k_i * inst->dt + inst->iyOld;
	FB_Integrator(&inst->integrator);
	inst->u = BON((BON(inst->e * inst->k_p) + inst->integrator.out));

	inst->iyOld = inst->u - (BON(inst->e * inst->k_p) + inst->integrator.out);
}
```

### Library Logical/Libraries/Library1 (ANSIC)

#### Library1.fun - Exported functions and function blocks
```iecst
{REDUND_ERROR} {REDUND_UNREPLICABLE} FUNCTION_BLOCK FB_Integrator (*TODO: Add your comment here*) (*$GROUP=User,$CAT=User,$GROUPICON=User.png,$CATICON=User.png*)
	VAR_INPUT
		in : {REDUND_UNREPLICABLE} REAL;
	END_VAR
	VAR_OUTPUT
		out : {REDUND_UNREPLICABLE} REAL;
	END_VAR
	VAR
		dt : {REDUND_UNREPLICABLE} REAL;
	END_VAR
END_FUNCTION_BLOCK

{REDUND_ERROR} {REDUND_UNREPLICABLE} FUNCTION_BLOCK FBMotor (*TODO: Add your comment here*) (*$GROUP=User,$CAT=User,$GROUPICON=User.png,$CATICON=User.png*)
	VAR_INPUT
		u : {REDUND_UNREPLICABLE} REAL;
	END_VAR
	VAR_OUTPUT
		w : {REDUND_UNREPLICABLE} REAL;
		phi : {REDUND_UNREPLICABLE} REAL;
	END_VAR
	VAR
		integrator : {REDUND_UNREPLICABLE} FB_Integrator;
		Tm : {REDUND_UNREPLICABLE} REAL;
		ke : {REDUND_UNREPLICABLE} REAL;
		dt : {REDUND_UNREPLICABLE} REAL;
	END_VAR
END_FUNCTION_BLOCK

{REDUND_ERROR} {REDUND_UNREPLICABLE} FUNCTION_BLOCK FB_Regulator (*TODO: Add your comment here*) (*$GROUP=User,$CAT=User,$GROUPICON=User.png,$CATICON=User.png*)
	VAR_INPUT
		e : {REDUND_UNREPLICABLE} REAL;
	END_VAR
	VAR_OUTPUT
		u : {REDUND_UNREPLICABLE} REAL;
	END_VAR
	VAR
		k_p : {REDUND_UNREPLICABLE} REAL;
		k_i : {REDUND_UNREPLICABLE} REAL;
		integrator : {REDUND_UNREPLICABLE} FB_Integrator;
		iyOld : {REDUND_UNREPLICABLE} REAL;
		max_abc_value : {REDUND_UNREPLICABLE} REAL;
		dt : {REDUND_UNREPLICABLE} REAL;
		x : {REDUND_UNREPLICABLE} REAL;
	END_VAR
END_FUNCTION_BLOCK
```

#### FB_Integrator.c
```c
#include <bur/plctypes.h>
#ifdef __cplusplus
	extern "C"
	{
#endif
	#include "Library1.h"
#ifdef __cplusplus
	};
#endif
/* TODO: Add your comment here */
void FB_Integrator(struct FB_Integrator* inst)
{
	inst->out = inst->in  + inst->out;

}
```

#### FBMotor.c
```c
#include <bur/plctypes.h>
#ifdef __cplusplus
	extern "C"
	{
#endif
	#include "Library1.h"
#ifdef __cplusplus
	};
#endif
/* TODO: Add your comment here */
void FBMotor(struct FBMotor* inst)
{
	inst->integrator.in = (inst->u/inst->ke - inst->w) * (inst->dt/inst->Tm);
	FB_Integrator(&inst->integrator);
	inst->w = inst->integrator.out;
	inst->integrator.in = inst->w * inst->dt;
	FB_Integrator(&inst->integrator);
	inst->phi = inst->integrator.out;
}
```

#### FB_Regulator.c
```c
#include <bur/plctypes.h>
#ifdef __cplusplus
	extern "C"
	{
#endif
	#include "Library1.h"
#ifdef __cplusplus
	};
#endif
/* TODO: Add your comment here */
void FB_Regulator(struct FB_Regulator* inst)
{
	float BON(float x)
	{
		if(x < 0)
		{
			if(x < -inst->max_abc_value)
				return -inst->max_abc_value;
			else
				return x;
		}
		else
		{
			if(x > inst->max_abc_value)
				return inst->max_abc_value;
			else
				return x;
		}

	}
	inst->integrator.in = inst->e * inst->k_i * inst->dt + inst->iyOld;
	FB_Integrator(&inst->integrator);
	inst->u = BON((BON(inst->e * inst->k_p) + inst->integrator.out));

	inst->iyOld = inst->u - (BON(inst->e * inst->k_p) + inst->integrator.out);
}
```

### Data object Logical/AxisApt (Apt)

#### AcpParTab.apt
```
AcoposParameterTable:
  Root Parameters:
    64201 = 4000 (Name=SERVO_V_MAX_OUTPUT, Unit=Units/s)  // Servo drive adjustment: Velocity at maximum output value
    109 = 24 (Name=SCALE_ENCOD_INCR)  // Encoder1: Encoder scaling: increments per encoder revolution
```

### Data object Logical/AxisInit (Ax)

#### AxInitAcp10.ax
```
InitParameter (Version=3.13.1, NcSwId=ACP10)
  ACP10AXIS_typ:
    dig_in:
      level:
        reference = ncACTIV_HI
        pos_hw_end = ncACTIV_HI
        neg_hw_end = ncACTIV_HI
        trigger1 = ncACTIV_HI
        trigger2 = ncACTIV_HI
    encoder_if:
      parameter:
        count_dir = ncSTANDARD
        scaling:
          load:
            units = 3000
            rev_motor = 1
    limit:
      parameter:
        v_pos = 7500.0
        v_neg = 7500.0
        a1_pos = 10000.0
        a2_pos = 10000.0
        a1_neg = 10000.0
        a2_neg = 10000.0
        t_jolt = 0.0
        t_in_pos = 0.0
        pos_sw_end = 8388607
        neg_sw_end = -8388608
        ds_warning = 500.0
        ds_stop = 50000.0
        a_stop = 1.0E+30
        dv_stop = 0.0
        dv_stop_mode = ncOFF
    controller:
      mode = ncPOSITION
      position:
        kv = 10.0
        tn = 0.0
        t_predict = 0.04
        t_total = 0.04
        p_max = 10000.0
        i_max = 0.0
      speed:
        kv = 2.0
        tn = 0.0
        t_filter = 0.0
        isq_filter1:
          type = ncOFF
          a0 = 0.0
          a1 = 0.0
          b0 = 0.0
          b1 = 0.0
          b2 = 0.0
          c0_par_id = 0
          c1_par_id = 0
        isq_filter2:
          type = ncOFF
          a0 = 0.0
          a1 = 0.0
          b0 = 0.0
          b1 = 0.0
          b2 = 0.0
          c0_par_id = 0
          c1_par_id = 0
        isq_filter3:
          type = ncOFF
          a0 = 0.0
          a1 = 0.0
          b0 = 0.0
          b1 = 0.0
          b2 = 0.0
          c0_par_id = 0
          c1_par_id = 0
      uf:
        type = ncLINEAR
        auto_config = ncMOTOR_PAR
        u0 = 0.0
        un = 0.0
        fn = 50.0
        k_f_slip = 0.0
      ff:
        torque_load = 0.0
        torque_pos = 0.0
        torque_neg = 0.0
        kv_torque = 0.0
        inertia = 0.0
        t_filter_a = 0.0
    move:
      stop:
        parameter[0]:
          decel_ramp = ncA_LIMIT
          controller = ncON
        parameter[1]:
          decel_ramp = ncA_LIMIT
          controller = ncON
        parameter[2]:
          decel_ramp = ncA_LIMIT
          controller = ncON
        parameter[3]:
          decel_ramp = ncA_LIMIT
          controller = ncON
        quickstop:
          decel_ramp = ncA_LIMIT
        drive_error:
          decel_ramp = ncA_LIMIT
      homing:
        parameter:
          s = 0
          v_switch = 6000.0
          v_trigger = 2000.0
          a = 10000.0
          mode = ncEND_SWITCH
          edge_sw = ncNEGATIVE
          start_dir = ncPOSITIVE
          trigg_dir = ncNEGATIVE
          ref_pulse = ncOFF
          fix_dir = ncOFF
          tr_s_block = 0.0
          torque_lim = 0.0
          ds_block = 0.0
          ds_stop = 0.0
      basis:
        parameter:
          v_pos = 4000.0
          v_neg = 4000.0
          a1_pos = 10000.0
          a2_pos = 10000.0
          a1_neg = 10000.0
          a2_neg = 10000.0
    message:
      text:
        parameter:
          format = ncBREAK
          columns = 80
          data_modul
```

### Data object Logical/acp10etxen (Ett)

- acp10etxen.ett (not shown)

### Package Logical/gAxis03obj - gAxis03obj

### Data object Logical/gAxis03obj/gAxis03a (Apt)

#### gAxis03a.apt
```
AcoposParameterTable:
  Root Parameters:
    230 = PCTRL_S_SET (Name=PCTRL_S_ACT_PARID)
    64201 = 546116.666666667 (Name=SERVO_V_MAX_OUTPUT)
```

### Data object Logical/gAxis03obj/gAxis03i (Ax)

#### gAxis03i.ax
```
InitParameter (Version=3.13.1, NcSwId=Acp10)
  ACP10AXIS_typ:
    dig_in:
      level:
        reference = ncACTIV_HI
        pos_hw_end = ncACTIV_HI
        neg_hw_end = ncACTIV_HI
        trigger1 = ncACTIV_HI
        trigger2 = ncACTIV_HI
    encoder_if:
      parameter:
        count_dir = ncSTANDARD
        scaling:
          load:
            units = 1000
            rev_motor = 1
    limit:
      parameter:
        v_pos = 10000
        v_neg = 10000
        a1_pos = 50000
        a2_pos = 50000
        a1_neg = 50000
        a2_neg = 50000
        t_jolt = 0
        t_in_pos = 0
        pos_sw_end = 2000000000
        neg_sw_end = -2000000000
        ds_warning = 500
        ds_stop = 1000
        a_stop = 1.0e30
        dv_stop = 0
        dv_stop_mode = ncOFF
    controller:
      mode = ncPOSITION
      position:
        kv = 50
        tn = 0
        t_predict = 0.01
        t_total = 0.01
        p_max = 1.0e30
        i_max = 0
      speed:
        kv = 2.0
        tn = 0
        t_filter = 0.0
        isq_filter1:
          type = ncOFF
          a0 = 0.0
          a1 = 0.0
          b0 = 0.0
          b1 = 0.0
          b2 = 0.0
          c0_par_id = 0
          c1_par_id = 0
        isq_filter2:
          type = ncOFF
          a0 = 0.0
          a1 = 0.0
          b0 = 0.0
          b1 = 0.0
          b2 = 0.0
          c0_par_id = 0
          c1_par_id = 0
        isq_filter3:
          type = ncOFF
          a0 = 0.0
          a1 = 0.0
          b0 = 0.0
          b1 = 0.0
          b2 = 0.0
          c0_par_id = 0
          c1_par_id = 0
      uf:
        type = ncLINEAR
        auto_config = ncMOTOR_PAR
        u0 = 0
        un = 0
        fn = 50.0
        k_f_slip = 0
      ff:
        torque_load = 0.0
        torque_pos = 0.0
        torque_neg = 0.0
        kv_torque = 0.0
        inertia = 0.0
        t_filter_a = 0.0
    move:
      stop:
        parameter[0]:
          decel_ramp = ncA_LIMIT
          controller = ncON
        parameter[1]:
          decel_ramp = ncA_LIMIT
          controller = ncON
        parameter[2]:
          decel_ramp = ncA_LIMIT
          controller = ncON
        parameter[3]:
          decel_ramp = ncA_LIMIT
          controller = ncON
        quickstop:
          decel_ramp = ncA_LIMIT
        drive_error:
          decel_ramp = ncA_LIMIT
      homing:
        parameter:
          s = 0
          v_switch = 5000
          v_trigger = 500
          a = 50000
          mode = ncEND_SWITCH
          edge_sw = ncPOSITIVE
          start_dir = ncPOSITIVE
          trigg_dir = ncPOSITIVE
          ref_pulse = ncOFF
          fix_dir = ncOFF
          tr_s_block = 0
          torque_lim = 0
          ds_block = 0
          ds_stop = 0
      basis:
        parameter:
          v_pos = 5000
          v_neg = 5000
          a1_pos = 50000
          a2_pos = 50000
          a1_neg = 50000
          a2_neg = 50000
    message:
      text:
        parameter:
          format = ncBREAK
          columns = 80
          data_modul = acp10etxen
```

### Program Logical/SDCAxisCtrl_X (ANSIC)

#### Main.c - Init, cyclic, exit code
```c
#include <bur/plctypes.h>

#ifdef _DEFAULT_INCLUDES
	#include <AsDefault.h>
#endif

void increase_counters(void);
void Homing(void);

void _INIT ProgramInit(void)
{
	//Устанваливаем типы SDC модулей
	AxisX_HW.EncIf1_Typ = ncSDC_ENC16;
	AxisX_HW.DiDoIf_Typ = ncSDC_DIDO;
	AxisX_HW.DrvIf_Typ = ncSDC_DRVSERVO16;

	//Устанавливаем имена переменных
	strcpy(AxisX_HW.EncIf1_Name, "AxisX_EncIf");
	strcpy(AxisX_HW.DrvIf_Name, "AxisX_DrvIf");
	strcpy(AxisX_HW.DiDoIf_Name, "AxisX_DiDoIf");

	//Устанавливаем входы готовности и нормальной работы
	AxisX_EncIf.iEncOK = 1;
	AxisX_DrvIf.iDrvOK = 1;
	AxisX_DrvIf.iStatusEnable = 1;
	AxisX_DiDoIf.iDriveReady = 1;

	fb_regulator.dt = 0.002;
	fb_regulator.k_i = 0.16;
	fb_regulator.k_p = 0.0064;
	fb_regulator.max_abc_value = 24.0;

	pwm_period = 200;
}

void _CYCLIC ProgramCyclic(void)
{
	increase_counters();
	AxisX_EncIf.iActTime = (INT)AsIOTimeCyclicStart();
	iPosHwEnd = axis_X.endswitch_a_reached;
	iNegHwEnd = axis_X.endswitch_b_reached;

	if(coil_powered == 1)
	{
		if(!Already_Homed)
		{
			Homing();
		}
		else
		{
			increase_counters();
			axis_X.reset_counter = 0;
			FB_Axis(&axis_X);
			coil_pwm_value = 32767;
			iPosHwEnd = axis_X.endswitch_a_reached;
			iNegHwEnd = axis_X.endswitch_b_reached;
			FB_Axis(&axis_X);

			fb_regulator.e = (AxisX_DrvIf.oSetPos*10)  - axis_X.speed;//oSetPos;
			FB_Regulator(&fb_regulator);

			axis_X.u = fb_regulator.u ;
			FB_Axis(&axis_X);}
	}
	else
	{
		coil_pwm_value = 0;
		fb_regulator.e = 0 ;
		FB_Regulator(&fb_regulator);
		axis_X.u = 0;
		FB_Axis(&axis_X);

	}
	// COUNTER1 = axis_X.counter

	//COUNTER2 += axis_X.counter - COUNTER1;
}

void increase_counters(void)
{
	AxisX_EncIf.iLifeCnt++;
	AxisX_DiDoIf.iLifeCntDriveEnable++;
	AxisX_DiDoIf.iLifeCntDriveReady++;
	AxisX_DiDoIf.iLifeCntNegHwEnd++;
	AxisX_DiDoIf.iLifeCntPosHwEnd++;
	AxisX_DiDoIf.iLifeCntReference++;
	AxisX_DrvIf.iLifeCnt++;
}

void Homing(void)
{
	increase_counters();
	coil_pwm_value = 32767;
	iPosHwEnd = axis_X.endswitch_a_reached;
	iNegHwEnd = axis_X.endswitch_b_reached;
	FB_Axis(&axis_X);

	fb_regulator.e = (AxisX_DrvIf.oSetPos * 10) - axis_X.speed;//oSetPos;
	FB_Regulator(&fb_regulator);

	axis_X.u = fb_regulator.u ;
	FB_Axis(&axis_X);
	if (iPosHwEnd)
	{
		coil_pwm_value = 0;
		fb_regulator.e = 0;
		FB_Regulator(&fb_regulator);
		axis_X.u = 0;
		FB_Axis(&axis_X);
		axis_X.reset_counter = 1;
		FB_Axis(&axis_X);
		if(k == 200)
		{
			Already_Homed = 1;
			FB_Axis(&axis_X);
		}
		k++;

	}

}

void _EXIT ProgramExit(void)
{
	// Insert code here

}
```

#### Variables.var - Local variables
```iecst
VAR
	min_task : INT := 7000;
	desired_speed : INT := 0;
	axis_X : FB_Axis;
	coil_powered : BOOL := FALSE;
	coil_pwm_value : {REDUND_UNREPLICABLE} INT := 200;
	fb_controller : FB_Controller;
	pwm_period : {REDUND_UNREPLICABLE} UINT := 200;
	Already_Homed : BOOL := FALSE;
	k : INT := 0;
	reset : BOOL := FALSE;
END_VAR
```

### Program Logical/ncsdcctrl (IEC)

#### ncsdcctrlCyclic.st
```iecst
PROGRAM _CYCLIC

(* ### BEGIN gAxis05 ### *)

(* life counter emulation of digital inputs *)
      gAxis05_DiDoIf.iLifeCntReference := gAxis05_DiDoIf.iLifeCntReference + 1;
      gAxis05_DiDoIf.iLifeCntNegHwEnd  := gAxis05_DiDoIf.iLifeCntNegHwEnd  + 1;
      gAxis05_DiDoIf.iLifeCntPosHwEnd  := gAxis05_DiDoIf.iLifeCntPosHwEnd  + 1;

(* default function model of ACOPOSmicro: convert absolute steps to delta steps - overflow save delta calculation *)
      gAxis05_MotorStep0 := gAxis05_DrvIf.oSetPos - gAxis05_oSetPosOld;
      gAxis05_oSetPosOld := gAxis05_DrvIf.oSetPos;

(* ### END gAxis05 ### *)

END_PROGRAM
```

#### ncsdcctrlInit.st
```iecst
PROGRAM _INIT

(* ### BEGIN gAxis05 ### *)

(* initialize general interfaces *)
      gAxis05.size := gAxis05.size;
      gAxis05_HW.DrvIf_Typ := ncSDC_DRVSM16;
      brsstrcpy( ADR(gAxis05_HW.DrvIf_Name[0]), ADR('gAxis05_DrvIf') );
      gAxis05_HW.DiDoIf_Typ := ncSDC_DIDO;
      brsstrcpy( ADR(gAxis05_HW.DiDoIf_Name[0]), ADR('gAxis05_DiDoIf') );
      gAxis05_HW.EncIf1_Typ := ncSDC_ENC16;
      brsstrcpy( ADR(gAxis05_HW.EncIf1_Name[0]), ADR('gAxis05_EncIf1') );
      gAxis05_EncIf1.iLifeCnt := gAxis05_EncIf1.iLifeCnt;

(* initialize old-value for delta step calculation *)
      gAxis05_oSetPosOld := gAxis05_DrvIf.oSetPos;

(* ### END gAxis05 ### *)

END_PROGRAM
```

#### ncsdcctrl.var
```iecst
VAR
	gAxis05_oSetPosOld : INT := 0;
END_VAR
```

### Package Logical/gAxis05obj - gAxis05obj

### Data object Logical/gAxis05obj/gAxis05a (Apt)

#### gAxis05a.apt
```
AcoposParameterTable:
  Root Parameters:
    64232 = 51200 (Name=SM_SCALE_STEP)
    64233 = 1000 (Name=SM_SCALE_LOAD_UNITS)
    64234 = 1 (Name=SM_SCALE_LOAD_MOTREV)
    109 = 1024 (Name=SCALE_ENCOD_INCR)
```

### Data object Logical/gAxis05obj/gAxis05i (Ax)

#### gAxis05i.ax
```
InitParameter (Version=3.13.1, NcSwId=Acp10)
  ACP10AXIS_typ:
    dig_in:
      level:
        reference = ncACTIV_HI
        pos_hw_end = ncACTIV_LO
        neg_hw_end = ncACTIV_LO
        trigger1 = ncACTIV_HI
        trigger2 = ncACTIV_LO + ncQUICKSTOP
    encoder_if:
      parameter:
        count_dir = ncSTANDARD
        scaling:
          load:
            units = 1000
            rev_motor = 1
    limit:
      parameter:
        v_pos = 10000
        v_neg = 10000
        a1_pos = 50000
        a2_pos = 50000
        a1_neg = 50000
        a2_neg = 50000
        t_jolt = 0
        t_in_pos = 0
        pos_sw_end = 2000000000
        neg_sw_end = -2000000000
        ds_warning = 500
        ds_stop = 1000
        a_stop = 1.0e30
        dv_stop = 0
        dv_stop_mode = ncOFF
    controller:
      mode = ncPOSITION
      position:
        kv = 50
        tn = 0
        t_predict = 0.01
        t_total = 0.01
        p_max = 1.0e30
        i_max = 0
      speed:
        kv = 2.0
        tn = 0
        t_filter = 0.0
        isq_filter1:
          type = ncOFF
          a0 = 0.0
          a1 = 0.0
          b0 = 0.0
          b1 = 0.0
          b2 = 0.0
          c0_par_id = 0
          c1_par_id = 0
        isq_filter2:
          type = ncOFF
          a0 = 0.0
          a1 = 0.0
          b0 = 0.0
          b1 = 0.0
          b2 = 0.0
          c0_par_id = 0
          c1_par_id = 0
        isq_filter3:
          type = ncOFF
          a0 = 0.0
          a1 = 0.0
          b0 = 0.0
          b1 = 0.0
          b2 = 0.0
          c0_par_id = 0
          c1_par_id = 0
      uf:
        type = ncLINEAR
        auto_config = ncMOTOR_PAR
        u0 = 0
        un = 0
        fn = 50.0
        k_f_slip = 0
      ff:
        torque_load = 0.0
        torque_pos = 0.0
        torque_neg = 0.0
        kv_torque = 0.0
        inertia = 0.0
        t_filter_a = 0.0
    move:
      stop:
        parameter[0]:
          decel_ramp = ncA_LIMIT
          controller = ncON
        parameter[1]:
          decel_ramp = ncA_LIMIT
          controller = ncON
        parameter[2]:
          decel_ramp = ncA_LIMIT
          controller = ncON
        parameter[3]:
          decel_ramp = ncA_LIMIT
          controller = ncON
        quickstop:
          decel_ramp = ncA_LIMIT
        drive_error:
          decel_ramp = ncA_LIMIT
      homing:
        parameter:
          s = 0
          v_switch = 5000
          v_trigger = 500
          a = 50000
          mode = ncDIRECT
          edge_sw = ncPOSITIVE
          start_dir = ncPOSITIVE
          trigg_dir = ncPOSITIVE
          ref_pulse = ncOFF
          fix_dir = ncOFF
          tr_s_block = 0
          torque_lim = 0
          ds_block = 0
          ds_stop = 0
      basis:
        parameter:
          v_pos = 5000
          v_neg = 5000
          a1_pos = 50000
          a2_pos = 50000
          a1_neg = 50000
          a2_neg = 50000
    message:
      text:
        parameter:
          format = ncBREAK
          columns = 80
          data_modul = acp10etxen
```

Listed in the project but not available here: Logical/Global.typ, Logical/Libraries/Library1/Types.typ, Logical/Libraries/Library1/Constants.var, Logical/Types.typ, Logical/ncsdcctrl/ncsdcctrl.typ
